(* Logix 5000 project; controller TCP vendor 1 type 14 code 178 rev 35.12; software revision 35.01 *)

TASK MainTask (continuous, watchdog 500 ms) : MainProgram, TCP_Connection
TASK SafetyTask (periodic, rate 20 ms, priority 10, watchdog 20 ms, safety) : SafetyProgram

MODULES
   Local : vendor 1 type 14 code 178 (Compact 0, rev 35.12)
END_MODULES

TYPE MSG_CreateParameters :
STRUCT
   Type : DINT;   // 1 - TCP ; 2 - UPD
   Addr : MSG_SockAddr;   // Address for the Socket
END_STRUCT
END_TYPE

TYPE MSG_OpenConnectionParameters :
STRUCT
   TimeOut : DINT;   // Timeout in milliseconds
   DestAddr : STRING;   // Hostname or IP adress (ex : 10.88.81.10?port=2813 OR name?port=2813)
END_STRUCT
END_TYPE

TYPE MSG_ReadParameters :
STRUCT
   TimeOut : DINT;   // TimeOut in milliseconds
   BufLen : DINT;   // Number of bytes of data to receive
END_STRUCT
END_TYPE

TYPE MSG_ReadResponse :
STRUCT
   FromAddr : MSG_SockAddr;   // A user-defined structure that can contain the address of the device that sends UDP data. This structure is populated from the end device. For TCP or UDP with OpenConnection, this structure is not used and contains all zeros. The TCP connection conveys all remote address information
   BufLen : DINT;   // Contains the number of bytes of data received
   Buf : SINT[484];   // Contains the data. This number must be large enough to contain the maximum amount of data expected. For a standard connection, the maximum is SINT[484]. For a large connection, the maximum is SINT [3984].
END_STRUCT
END_TYPE

TYPE MSG_SockAddr :
STRUCT
   Family : INT;   // Adress Family Must be 2
   Port : INT;   // Port Number - If random needed use 0
   Addr : DINT;   // IP Address - Each Byte are separated for xxx.xxx.xxx.xxx
END_STRUCT
END_TYPE

TYPE MSG_WriteParameters :
STRUCT
   TimeOut : DINT;   // TimeOut in milliseconds
   ToAddr : MSG_SockAddr;   // Structure that contains the address to which to write UDP data. For TCP or UDP with OpenConnection, this structure is not used and contains all zeros. The TCP connection conveys all required remote address information.
   BufLen : DINT;   // Specify the number of bytes of data to write
   Buf : SINT[472];   // Contains the data. This number must be large enough to contain the maximum amount of data expected. For a standard connection, the maximum is SINT[472]. For a large connection, the maximum is SINT [3972].
END_STRUCT
END_TYPE

TYPE UDT_ACTION :   // Action
STRUCT
   Comp : BOOL;   // Action Completed
   OppComp : BOOL;   // Opposite Action Completed
   Clear : BOOL;   // Action is Clear to Go
   Cond_Clear : UDT_ACTION_CLEAR[32];   // Conditions & Texts for Clear (HMI & Supervisor)
   OutPwr : BOOL;   // Output Power For Action
   Cmd : BOOL;   // Action Command
   VirtualOut : BOOL;   // Action Output Request (Virtual )
   Out : BOOL;   // Action Output
   Mem : BOOL;   // Action Memory
   Fault : BOOL;   // Action Faulted
   ActionRequest : BOOL;   // Action Request
END_STRUCT
END_TYPE

TYPE UDT_ACTION_CLEAR :
STRUCT
   Used : BOOL;   // Condition used
   State : BOOL;   // State of the condition
   Text : STRING;   // Text of the condition for HMI & Supervisor
END_STRUCT
END_TYPE

TYPE UDT_BLINK :
STRUCT
   _250ms : BOOL;   // 250ms ON; 250ms OFF
   _500ms : BOOL;   // 500ms ON; 500ms OFF
   _1s : BOOL;   // 1s ON; 1s OFF
   Fast : BOOL;   // Fast Blinking
   Normal : BOOL;   // Normal Blinking
   Edge_1s : BOOL;   // Egde 1s
   Edge_100ms : BOOL;   // Edge 100ms
   Edge_5s : BOOL;   // Edge 5s
END_STRUCT
END_TYPE

TYPE UDT_COOL_DI :
STRUCT
   Load_Presence : BOOL;
   Fan1_CR : BOOL;
   Fan2_CR : BOOL;
END_STRUCT
END_TYPE

TYPE UDT_EDGES :
STRUCT
   Dir_Action : BOOL;   // Direct Action for Raising Edge
   Rev_Action : BOOL;   // Reverse Action for Raising Edge
   Auto_Mode : BOOL;   // Operating Mode Automatic Running for Raising Edge
   Auto_Mode_Switch : BOOL;   // Automatic Mode Switch for Raising Edge
   Manual_Mode_Switch : BOOL;   // Manual Mode Switch for Raising Edge
   Area_Gate_1 : BOOL;   // Area Gate 1 Closed & Locked
   Area_Gate_2 : BOOL;   // Area Gate 2 Closed & Locked
   Area_Gate_3 : BOOL;   // Area Gate 3 Closed & Locked
   Area_Gate_4 : BOOL;   // Area Gate 4 Closed & Locked
   Area_Gate_5 : BOOL;   // Area Gate 5 Closed & Locked
END_STRUCT
END_TYPE

TYPE UDT_FAULT_TREATMENT :
STRUCT
   SAF_DF : INT;   // Faults
   SAF_DF_COPY : INT;   // Fault Copy for Edge Detection
   FAULT_DF : INT[10];   // Faults
   FAULT_COPY : INT[10];   // Fault Copy for Edge Detection
   Level1_Fault_Present : BOOL;   // Level 1 Fault Present
   Level2_Fault_Present : BOOL;   // Level 2 Fault Present
   Level3_Fault_Present : BOOL;   // Level 3 Fault Present
   Level4_Fault_Present : BOOL;   // Level 4 Fault Present
   Fault_Presence : BOOL;   // Fault Presence
   Fault_Appearence : BOOL;   // Fault Appearence
   Treatment_Fault_Copy : BOOL;   // Treatment Fault Copy
   Treatment_Fault_Presence : BOOL;   // Treatment Fault Presence
   Treatment_Fault_Appearence : BOOL;   // Treatment Fault Appearence
END_STRUCT
END_TYPE

TYPE UDT_GEN_ACTION :
STRUCT
   Forcing_Acces_Door : UDT_ACTION;   // Forcing Acces Door for opening
END_STRUCT
END_TYPE

TYPE UDT_GEN_AI :   // Analog Inputs
STRUCT
   Spare : INT;
END_STRUCT
END_TYPE

TYPE UDT_GEN_DELAY :
STRUCT
   Encoding_Req : INT;   // GEN -- Delay Encoding Request
   Encoding_Checksum_Calc_Req : INT;   // GEN -- Delay Encoding Checksum Calculation Request
END_STRUCT
END_TYPE

TYPE UDT_GEN_DELAY_ON :
STRUCT
   Encoding_Req : BOOL;   // GEN -- Delay Encoding Request
   Encoding_Checksum_Calc_Req : BOOL;   // GEN -- Delay Encoding Checksum Calculation Request
END_STRUCT
END_TYPE

TYPE UDT_GEN_DI :   // Digital Inputs
STRUCT
   Reset_EStop : BOOL;   // SBHL19003 : Reset Emergency Stop PB
   Power_ON : BOOL;   // KA8501 : Power ON
   Air_Cond_Temp_OK : BOOL;   // P3601 : Cabinet Air Temperature
   WL_Alarm : BOOL;   // CR241 : Water Loop Alarm Relay
   Auto_Switch : BOOL;   // SB19601 : Selector Auto
   Manual_Switch : BOOL;   // SB19601 : Selector Manu
   Silence_Horn : BOOL;   // SB19602 : Silence Horn
   Reset : BOOL;   // SB19603 : Reset Default
   Reset_Light : BOOL;   // SBHL20702 : Reset Light Curtain
   STORAGE : UDT_STO_DI[64];
   COOL : UDT_COOL_DI[64];
   PC_KTP_Switch : BOOL;   // 0=PC ; 1=KTP
   Direct_Action_Pb : BOOL;   // Direct Action Pushbutton
   Reverse_Action_Pb : BOOL;   // Reverse Action Pushbutton
END_STRUCT
END_TYPE

TYPE UDT_GEN_DO_LIGHT :   // Digital Outputs (Light & Horn)
STRUCT
   Horn : BOOL;   // H24501/H24601 : Horn
   Column_Green : BOOL;   // HL24502/HL24602 : Column Green Light Automatic / Ready
   Column_Red : BOOL;   // HL24503/HL24603 : Column Red Light Critical Event / Fault
   Column_Yellow : BOOL;   // HL24504/HL24604 : Column Yellow Light Manual / Warning
   Column_Blue : BOOL;   // HL24505/HL24605 : Column Blue Light External Help Request
   Column_White : BOOL;   // HL24506/HL24606 : Column White Light Set Up Mode
   Reset_Fault_Light : BOOL;   // PBL19603 : Reset Fault Light
END_STRUCT
END_TYPE

TYPE UDT_GEN_FAULT :
STRUCT
   Gen_Cab_EStop : BOOL;   // Fault : GEN - General Cabinet Estop
   Power_ON : BOOL;   // Fault General Start
   UPS_ON : BOOL;   // Fault UPS ON
   Air_Cond_OK : BOOL;   // Fault Exchanger and Air Temperature Control
   Area_Closed : BOOL;
   PC_EStop : BOOL;   // Fault GEN - Supervisory PC Estop
   UPS_Alarm : BOOL;   // Fault UPS: GEN - UPS Alarm
   UPS_Bat_Disch : BOOL;   // Fault UPS: GEN - Battery is Discharging
   UPS_Batt_Low : BOOL;   // Fault UPS: GEN - Battery Low!!
   UPS_Bypassed : BOOL;   // Fault UPS: GEN - UPS Bypassed
   UPS_Ext_Bypassed : BOOL;   // Fault GEN - External Bypass
   PLC_StopMode : BOOL;   // Fault GEN - PLC in STOP
   Manual_Mode : BOOL;   // Warning: GEN - Periph in Manual Mode
   OPTP_Calculation : BOOL;   // Fault OPTP : Calculation Fault
   OPTP_EL_TR_NRdy : BOOL;   // Fault OPTP EL : Start or Dest Cell not ready for Transfer
   Sfty_Sign_Not_Locked : BOOL;   // Fault GEN - Safety not Locked - Safety Program is not Protected
   Sfty_Sign_Missing : BOOL;   // Fault GEN - Safety Missing Signature - Generate Safety Signature before Locking Task
   Sfty_Sign_Mismatch : BOOL;   // Fault GEN - Safety Signature Mismatch - Safety Program has been Modified
   Com_PC_Loading : BOOL;   // Fault GEN - Communication Fault with PC Supervisory on Loading Side
   Com_PC_Unloading : BOOL;   // Fault GEN - Communication Fault with PC Supervisory on Unloading Side
   Encoding_Error : BOOL;   // Fault GEN - L/U Cell - Encoding Error
   Com_PLC_NANO1 : BOOL;   // Error communication with NANO1
   Com_PLC_NANO2 : BOOL;   // Error communication with NANO2
   Com_PLC_CRYO : BOOL;   // Error communication with CRYO
   Com_PLC_TEMP1 : BOOL;   // Error communication with TEMPER 1
   Com_PLC_TEMP2 : BOOL;   // Error communication with TEMPER 2
   Com_PLC_TEMP3 : BOOL;   // Error communication with TEMPER 3
   Com_PLC_TEMP4 : BOOL;   // Error communication with TEMPER 4
   Com_PLC_TEMP5 : BOOL;   // Error communication with TEMPER 5
   WL_Alarm : BOOL;   // Water Loop : Alarm Relay
   Load_Rejected_Qty_Max : BOOL;   // Load rejected Quantity Max for the Recipe
   Load_Rejected_Qty_Min : BOOL;   // Load rejected Quantity Min for the Recipe
   Load_Rejected_Error_Heat_Recipe : BOOL;   // Load rejected Error in the Step of the Heating Recipe (Temperature must be the same between Ramp and Step after)
   Load_Rejected_Weight_too_heavy : BOOL;   // Load Rejected Error on Total Weight too heavy > 100Kg - 220lbs
   TManager_GetCaution_Error : BOOL;   // T-Manager - GetCaution Request Error
   TManager_GetInstruction_Error : BOOL;   // T-Manager - GetInstruction Request Error
   TManager_TestRunBefore_Error : BOOL;   // T-Manager - Test Run Before Request Error
   TManager_Download_Recipe_Error : BOOL;   // T-Manager - Download Recipe Request Error
   TManager_Insert_Error : BOOL;   // T-Manager - Insert Load Request Error
   TManager_Update_Data_Load_Error : BOOL;   // T-Manager - Update data Load Request Error
   Load_Rejected_Error_Heat_Step_Type : BOOL;   // Load Rejected Error Wrong Type of the Step of the Recipe (Heating cell & Quench )
   Load_Rejected_Miss_Times : BOOL;   // Load Rejected Error Miss times on the Recipe
   Waiting_Transfer_Timeout : BOOL;   // Next order is not in progress - miss conditions
   Miss_Start_Cell_Cond : BOOL;   // Next order is not in progress - Miss Start Cell condition
   Miss_Dest_Cell_Cond : BOOL;   // Next order is not in progress - Miss Dest Cell condition
   Miss_EL_Order_Auth : BOOL;   // Next order is not in progress - Miss Authorization Execution External Loader
END_STRUCT
END_TYPE

TYPE UDT_GEN_FAULT_DELAY :
STRUCT
   Gen_Cab_EStop : INT;   // Fault : GEN - General Cabinet Estop
   Power_ON : INT;   // Fault General Start
   UPS_ON : INT;   // Fault UPS ON
   Air_Cond_OK : INT;   // Fault Exchanger and Air Temperature Control
   Area_Closed : INT;   // Fault GEN - Area Access Door Closed
   PC_EStop : INT;   // Fault GEN - Supervisory PC Estop
   UPS_Alarm : INT;   // Fault UPS: GEN - UPS Alarm
   UPS_Bat_Disch : INT;   // Fault UPS: GEN - Battery is Discharging
   UPS_Batt_Low : INT;   // Fault UPS: GEN - Battery Low!!
   UPS_Bypassed : INT;   // Fault UPS: GEN - UPS Bypassed
   UPS_Ext_Bypassed : INT;   // Fault GEN - External Bypass
   PLC_StopMode : INT;   // Fault GEN - PLC in STOP
   Manual_Mode : INT;   // Warning: GEN - Nano in Manual Mode
   OPTP_Calculation : INT;   // Fault OPTP : Calculation Fault
   OPTP_EL_TR_NRdy : INT;   // Fault OPTP EL : Start or Dest Cell not ready for Transfer
   Sfty_Sign_Not_Locked : INT;   // Fault GEN - Safety not Locked - Safety Program is not Protected
   Sfty_Sign_Missing : INT;   // Fault GEN - Safety Missing Signature - Generate Safety Signature before Locking Task
   Sfty_Sign_Mismatch : INT;   // Fault GEN - Safety Signature Mismatch - Safety Program has been Modified
   Com_PC_Loading : INT;   // Fault GEN - Communication Fault with PC Supervisory on Loading Side
   Com_PC_Unloading : INT;   // Fault GEN - Communication Fault with PC Supervisory on Unloading Side
   Encoding_Error : INT;   // Fault GEN - L/U Cell - Encoding Error
   Com_Error_Send_Load_PLC_NANO1 : INT;   // Fault GEN - Error on the Send data for Load to the NANO1
   Timeout_Recv_Cyclic_PLC_NANO1 : INT;   // Fault GEN - Time out receiving data from PLC NANO1
   Com_Error_Send_Load_PLC_NANO2 : INT;   // Fault GEN - Error on the Send data for Load to the NANO2
   Timeout_Recv_Cyclic_PLC_NANO2 : INT;   // Fault GEN - Time out receiving data from PLC NANO2
   WL_Alarm : INT;
END_STRUCT
END_TYPE

TYPE UDT_GEN_FAULT_ETHIP :
STRUCT
   RemIO : BOOL;   // Ethernet IP : Rem IO
   x1 : BOOL;
   x2 : BOOL;
   x3 : BOOL;
   x4 : BOOL;
   E12401_MAIN : BOOL;
   E12501_MAIN : BOOL;
   X26001_MAIN : BOOL;   // Ethernet IP : X26001-Armblock
   X26002_MAIN : BOOL;   // Ethernet IP : X26001-Armblock
   X26101_MAIN : BOOL;   // Ethernet IP : X26101-Armblock
   X26201_MAIN : BOOL;   // Ethernet IP : X26201-Armblock
   X26301_MAIN : BOOL;   // Ethernet IP : X26301-Armblock
   X26401_MAIN : BOOL;   // Ethernet IP : X26401-Armblock (Water Loop)
   A6001_MAIN : BOOL;   // Ethernet IP : VFD A6001 - External Loader - Translation
   A6101_MAIN : BOOL;   // Ethernet IP : VFD A6001 - External Loader - Forks
   A6201_MAIN : BOOL;   // Ethernet IP : VFD A6001 - External Loader - Lifting
   A11201_FORTRESS : BOOL;   // Ethernet IP : FORTRESS A11201
   A11301_FORTRESS : BOOL;   // Ethernet IP : FORTRESS A11301
   E14201_STRATIX : BOOL;
   X26301_WL : BOOL;   // Ethernet IP : X26001-Armblock (Water Loop)
   Nano1 : BOOL;   // Ethernet IP : PLC Nano1
   Nano2 : BOOL;   // Ethernet IP : PLC Nano 2
   Cryo : BOOL;   // Ethernet IP : PLC Cryo
   Temper1 : BOOL;   // Ethernet IP : PLC Temper 1
   Temper2 : BOOL;   // Ethernet IP : PLC Temper 2
   Temper3 : BOOL;   // Ethernet IP : PLC Temper 3
   Temper4 : BOOL;   // Ethernet IP : PLC Temper 4
END_STRUCT
END_TYPE

TYPE UDT_GEN_FAULT_SAFETY :
STRUCT
   Estop : BOOL;   // GEN -EStop OK
   MCRA_ON : BOOL;   // GEN - MCR 1A/2A (Emergency Stop)
   SCRA_ON : BOOL;   // GEN - SCR 1A/2A
   SCRB_ON : BOOL;   // GEN - SCR 1B/2B
   SCRC_ON : BOOL;   // GEN - SCR 1C/2C
   Sfty_Ack_Req : BOOL;   // GEN Fault -- Safety Acknowledge Requested
END_STRUCT
END_TYPE

TYPE UDT_GEN_INFO :
STRUCT
   Normal_Supply : BOOL;   // GEN -- Normal Supply
   UPS_Supply : BOOL;   // GEN -- Saved Supply
   Normal_Volt_Flt_Mem : BOOL;   // GEN -- Normal Voltage presence Fault Memory
   KTP_Manual_Cmd_Auth : BOOL;   // GEN -- KTP Manual Command Authorization
   Init_Cond : BOOL;   // GEN -- Initial Conditions for Auto Mode
   Out_Oper_Mode : BOOL;   // GEN -- Conditions for Switching to Out of Operation Mode
   Stop_Oper_Mode : BOOL;   // GEN -- Stop Operation Mode
   No_Motion_for_Door_Access : BOOL;   // GEN - No Motion for Door Access
   No_Motion_EL : BOOL;   // External Loader : No motion
   No_Motion_LD : BOOL;   // Loading : No Motion
   No_Motion_UL : BOOL;   // Unloading : No Motion
   No_Motion_Cool : BOOL;   // Cooling : No Motion
   No_Motion_NANO : BOOL;   // NANO : No Motion (By dialogue)
   No_Motion_TEMP : BOOL;   // TEMPER : No Motion (By dialogue)
   No_Motion_CRYO : BOOL;   // CRYO : No Motion (By dialogue)
   Access_Request : BOOL;   // Request for access to the outer peripheral zone
   Access_Authorized : BOOL;   // Acces Authorized
   Access_OK : BOOL;   // Acces OK : Solenoid Active
   Cond_Auto_Mode : UDT_ACTION;   // Init Conditions for Auto Mode
   Cond_Auto_Mode_State : DINT;   // state for supervisory
   Cond_Auto_Mode_Used : DINT;   // Used for Supervisory
END_STRUCT
END_TYPE

TYPE UDT_GEN_MEAS :
STRUCT
   Spare : REAL;
END_STRUCT
END_TYPE

TYPE UDT_GEN_RUNNING_TIME :
STRUCT
   Spare : DINT;
END_STRUCT
END_TYPE

TYPE UDT_ID_READER :
STRUCT
   INPUT : UDT_ID_READER_IN;
   OUTPUT : UDT_ID_READER_OUT;
END_STRUCT
END_TYPE

TYPE UDT_ID_READER_IN :
STRUCT
   Sequence_Low : SINT;
   Sequence_High : SINT;
   LUID_Low : SINT;
   LUID_High : SINT;
   Bit_Counf_of_ID : SINT;
   Zero_Padding : SINT;
   ID_Data_bytes : SINT[32];
END_STRUCT
END_TYPE

TYPE UDT_ID_READER_OUT :
STRUCT
   Led_Control : BOOL;
   Beep : BOOL;
END_STRUCT
END_TYPE

TYPE UDT_OPERATING_MODE :
STRUCT
   Out_of_Operation : BOOL;   // Out of Operation Mode
   Init_Missing_Cond : BOOL;   // Operating Mode Initiales Conditions Missing
   Origin : BOOL;   // Operating Mode Origine
   Waiting_Cycle_Start : BOOL;   // Operating Mode Waiting for Cycle Start
   Manual : BOOL;   // Operating Mode Manual
   Auto : BOOL;   // Operating Mode Automatic Running
END_STRUCT
END_TYPE

TYPE UDT_OPTP_BUFFER :
STRUCT
   Buffer : SINT[5000];
   Lenght : DINT;
   New_Data : BOOL;
END_STRUCT
END_TYPE

TYPE UDT_OPTP_RECV_CONTROL :
STRUCT
   New_TCP_Data : BOOL;
   New_Frame_Complete : BOOL;
END_STRUCT
END_TYPE

TYPE UDT_STO_DI :
STRUCT
   Load_Presence_Physical : BOOL;   // Physical Presence on Storage
END_STRUCT
END_TYPE

VAR_GLOBAL   (* controller tags *)
   Destination_Element_Read_Request : MSG_ReadResponse := (FromAddr.Family := 2, Buf[0] := 107, Buf[1] := 99, Buf[2] := 111, Buf[9] := 1, Buf[12] := 107, Buf[13] := 99, Buf[14] := 111, Buf[21] := 3, Buf[25] := 1, Buf[29] := 1, Buf[34] := 15, Buf[35] := -125, Buf[36] := -20, Buf[37] := -78, Buf[38] := 50, Buf[39] := 54, Buf[40] := 48, Buf[41] := 51, Buf[42] := 48, Buf[43] := 52, Buf[44] := 48, Buf[45] := 53, Buf[46] := 48, Buf[61] := 3, Buf[63] := -115, Buf[64] := 23, Buf[65] := 112, Buf[66] := 19, Buf[67] := -119, Buf[75] := 48, Buf[76] := 7, Buf[77] := -47, Buf[79] := 60, Buf[80] := 107, Buf[81] := 99, Buf[82] := 111, Buf[89] := 3, Buf[91] := 1, Buf[92] := -20, Buf[93] := -95, Buf[94] := 50, Buf[95] := 54, Buf[96] := 48, Buf[97] := 51, Buf[98] := 48, Buf[99] := 52, Buf[100] := 48, Buf[101] := 51, Buf[102] := 51, Buf[117] := 93, Buf[119] := -115, Buf[120] := 2, Buf[121] := 89, Buf[122] := 19, Buf[123] := -119, Buf[126] := 4, Buf[127] := -52, Buf[130] := 5, Buf[131] := 8,
        Buf[132] := 7, Buf[133] := -41, Buf[135] := 60, Buf[136] := 107, Buf[137] := 99, Buf[138] := 111, Buf[145] := 3, Buf[147] := 2, Buf[148] := 107, Buf[149] := 99, Buf[150] := 111, Buf[157] := 3, Buf[159] := 2, Buf[160] := -20, Buf[161] := -95, Buf[162] := 50, Buf[163] := 54, Buf[164] := 48, Buf[165] := 51, Buf[166] := 48, Buf[167] := 52, Buf[168] := 48, Buf[169] := 51, Buf[170] := 51, Buf[185] := 93, Buf[187] := -115, Buf[188] := 2, Buf[189] := 89, Buf[190] := 19, Buf[191] := -119, Buf[194] := 5, Buf[195] := 59, Buf[198] := 5, Buf[199] := 119, Buf[200] := 7, Buf[201] := -41, Buf[203] := 60, Buf[204] := 107, Buf[205] := 99, Buf[206] := 111, Buf[213] := 3, Buf[215] := 3, Buf[216] := 107, Buf[217] := 99, Buf[218] := 111, Buf[225] := 3, Buf[227] := 3, Buf[229] := 4, Buf[233] := 4, Buf[238] := 15, Buf[239] := -125, Buf[240] := -20, Buf[241] := -95, Buf[242] := 50, Buf[243] := 54, Buf[244] := 48, Buf[245] := 51, Buf[246] := 48, Buf[247] := 52, Buf[248] := 48,
        Buf[249] := 51, Buf[250] := 51, Buf[265] := 93, Buf[267] := -115, Buf[268] := 2, Buf[269] := 89, Buf[270] := 19, Buf[271] := -119, Buf[274] := 9, Buf[275] := -13, Buf[278] := 10, Buf[279] := 47, Buf[280] := 7, Buf[281] := -41, Buf[283] := 60, Buf[284] := 107, Buf[285] := 99, Buf[286] := 111, Buf[293] := 3, Buf[295] := 4, Buf[297] := 5, Buf[301] := 5, Buf[306] := 15, Buf[307] := -125, Buf[308] := -20, Buf[309] := -95, Buf[310] := 50, Buf[311] := 54, Buf[312] := 48, Buf[313] := 51, Buf[314] := 48, Buf[315] := 52, Buf[316] := 48, Buf[317] := 51, Buf[318] := 51, Buf[333] := 93, Buf[335] := -115, Buf[336] := 2, Buf[337] := 89, Buf[338] := 19, Buf[339] := -119, Buf[342] := 13, Buf[343] := -50, Buf[346] := 14, Buf[347] := 10, Buf[348] := 7, Buf[349] := -41, Buf[351] := 60, Buf[352] := 107, Buf[353] := 99, Buf[354] := 111, Buf[361] := 3, Buf[363] := 5, Buf[365] := 6, Buf[369] := 6, Buf[374] := 15, Buf[375] := -125, Buf[376] := -20, Buf[377] := -95, Buf[378] := 50,
        Buf[379] := 54, Buf[380] := 48, Buf[381] := 51, Buf[382] := 48, Buf[383] := 52, Buf[384] := 48, Buf[385] := 51, Buf[386] := 51, Buf[401] := 93, Buf[403] := -115, Buf[404] := 2, Buf[405] := 89, Buf[406] := 19, Buf[407] := -119, Buf[410] := 14, Buf[411] := 25, Buf[414] := 14, Buf[415] := 85, Buf[416] := 7, Buf[417] := -41, Buf[419] := 60, Buf[420] := 107, Buf[421] := 99, Buf[422] := 111, Buf[429] := 3, Buf[431] := 6, Buf[433] := 7, Buf[437] := 7, Buf[442] := 15, Buf[443] := -125, Buf[444] := -20, Buf[445] := -95, Buf[446] := 50, Buf[447] := 54, Buf[448] := 48, Buf[449] := 51, Buf[450] := 48, Buf[451] := 52, Buf[452] := 48, Buf[453] := 51, Buf[454] := 51, Buf[469] := 93, Buf[471] := -115, Buf[472] := 2, Buf[473] := 89, Buf[474] := 19, Buf[475] := -119, Buf[478] := 15, Buf[479] := -31, Buf[482] := 16, Buf[483] := 29);
   Destination_Element_Write_Request : DINT := 48;   // Lenght of the Data written
   Instance_OPTP : DINT := 21276;
   MSG_Create_Socket : MESSAGE;
        MessageParameters(ServiceCode := 16#004b, LocalElement := Source_Element_Create_Socket, DestinationTag := Instance_OPTP, ...)
   MSG_Delete_All_Socket : MESSAGE;
        MessageParameters(ServiceCode := 16#0051, ...)
   MSG_Open_Connection : MESSAGE;
        MessageParameters(ServiceCode := 16#004c, LocalElement := Source_Element_Open_Connection, ...)
   MSG_Read_Request : MESSAGE;
        MessageParameters(ServiceCode := 16#004d, LocalElement := Source_Element_Read_Request, DestinationTag := Destination_Element_Read_Request, ...)
   MSG_Write_Request : MESSAGE;
        MessageParameters(ServiceCode := 16#004e, LocalElement := Source_Element_Write_Request, DestinationTag := Destination_Element_Write_Request, ...)
   Source_Element_Create_Socket : MSG_CreateParameters := (Type := 1, Addr.Family := 2, Addr.Port := 10002);   // Source parameters for MSG Create Socket
   Source_Element_Open_Connection : MSG_OpenConnectionParameters := (TimeOut := 5000, DestAddr := '192.120.0.203?port=5010$00');
   Source_Element_Read_Request : MSG_ReadParameters := (TimeOut := 3000, BufLen := 484);
   Source_Element_Write_Request : MSG_WriteParameters := (TimeOut := 5000, BufLen := 1, Buf[0] := 104, Buf[1] := 101, Buf[2] := 108, Buf[3] := 108, Buf[4] := 111);
END_VAR

PROGRAM MainProgram   (* main routine MainRoutine *)

ROUTINE MainRoutine   (* ladder *)
END_ROUTINE
END_PROGRAM

PROGRAM SafetyProgram   (* main routine MainRoutine, safety *)

ROUTINE MainRoutine   (* ladder *)
END_ROUTINE
END_PROGRAM

PROGRAM TCP_Connection   (* main routine Main *)
VAR
   buff_ind : DINT;
   Buff_ok : BOOL;
   Check_Buflenght : BOOL;
   Connection_Ok : BOOL := 1;
   Element_Read_buffer : SINT[5000];
   ind : DINT := 1;
   ONS : BOOL[32];
   Open_started : BOOL;
   OPTP_Data_RCV : UDT_OPTP_BUFFER := (Buffer[0] := 107, Buffer[1] := 99, Buffer[2] := 111, Buffer[9] := 3, Buffer[12] := 107, Buffer[13] := 99, Buffer[14] := 111, Buffer[21] := 3, Buffer[24] := -20, Buffer[25] := -78, Buffer[26] := 50, Buffer[27] := 54, Buffer[28] := 48, Buffer[29] := 51, Buffer[30] := 48, Buffer[31] := 52, Buffer[32] := 48, Buffer[33] := 53, Buffer[34] := 48, Buffer[49] := 3, Buffer[51] := -115, Buffer[52] := 23, Buffer[53] := 112, Buffer[54] := 19, Buffer[55] := -119, Buffer[63] := 48, Buffer[64] := 7, Buffer[65] := -47, Buffer[67] := 60, Buffer[68] := 107, Buffer[69] := 99, Buffer[70] := 111, Buffer[77] := 3, Buffer[79] := 1, Buffer[80] := 107, Buffer[81] := 99, Buffer[82] := 111, Buffer[89] := 3, Buffer[91] := 1, Buffer[92] := -20, Buffer[93] := -95, Buffer[94] := 50, Buffer[95] := 54, Buffer[96] := 48, Buffer[97] := 51, Buffer[98] := 48, Buffer[99] := 52, Buffer[100] := 48, Buffer[101] := 51, Buffer[102] := 51, Buffer[117] := 93, Buffer[119] := -115, Buffer[120] := 2, Buffer[121] := 89, Buffer[122] := 19, Buffer[123] := -119, Buffer[126] := 4, Buffer[127] := -52, Buffer[130] := 5, Buffer[131] := 8,
        Buffer[132] := 7, Buffer[133] := -41, Buffer[135] := 60, Buffer[136] := 107, Buffer[137] := 99, Buffer[138] := 111, Buffer[145] := 3, Buffer[147] := 2, Buffer[148] := 107, Buffer[149] := 99, Buffer[150] := 111, Buffer[157] := 3, Buffer[159] := 2, Buffer[160] := -20, Buffer[161] := -95, Buffer[162] := 50, Buffer[163] := 54, Buffer[164] := 48, Buffer[165] := 51, Buffer[166] := 48, Buffer[167] := 52, Buffer[168] := 48, Buffer[169] := 51, Buffer[170] := 51, Buffer[185] := 93, Buffer[187] := -115, Buffer[188] := 2, Buffer[189] := 89, Buffer[190] := 19, Buffer[191] := -119, Buffer[194] := 5, Buffer[195] := 59, Buffer[198] := 5, Buffer[199] := 119, Buffer[200] := 7, Buffer[201] := -41, Buffer[203] := 60, Buffer[204] := 107, Buffer[205] := 99, Buffer[206] := 111, Buffer[213] := 3, Buffer[215] := 3, Buffer[216] := 107, Buffer[217] := 99, Buffer[218] := 111, Buffer[225] := 3, Buffer[227] := 3, Buffer[228] := -20, Buffer[229] := -95, Buffer[230] := 50, Buffer[231] := 54, Buffer[232] := 48, Buffer[233] := 51, Buffer[234] := 48, Buffer[235] := 52, Buffer[236] := 48, Buffer[237] := 51, Buffer[238] := 51, Buffer[253] := 93, Buffer[255] := -115,
        Buffer[256] := 2, Buffer[257] := 89, Buffer[258] := 19, Buffer[259] := -119, Buffer[262] := 9, Buffer[263] := -13, Buffer[266] := 10, Buffer[267] := 47, Buffer[268] := 7, Buffer[269] := -41, Buffer[271] := 60, Buffer[272] := 107, Buffer[273] := 99, Buffer[274] := 111, Buffer[281] := 3, Buffer[283] := 4, Buffer[284] := 107, Buffer[285] := 99, Buffer[286] := 111, Buffer[293] := 3, Buffer[295] := 4, Buffer[296] := -20, Buffer[297] := -95, Buffer[298] := 50, Buffer[299] := 54, Buffer[300] := 48, Buffer[301] := 51, Buffer[302] := 48, Buffer[303] := 52, Buffer[304] := 48, Buffer[305] := 51, Buffer[306] := 51, Buffer[321] := 93, Buffer[323] := -115, Buffer[324] := 2, Buffer[325] := 89, Buffer[326] := 19, Buffer[327] := -119, Buffer[330] := 13, Buffer[331] := -50, Buffer[334] := 14, Buffer[335] := 10, Buffer[336] := 7, Buffer[337] := -41, Buffer[339] := 60, Buffer[340] := 107, Buffer[341] := 99, Buffer[342] := 111, Buffer[349] := 3, Buffer[351] := 5, Buffer[352] := 107, Buffer[353] := 99, Buffer[354] := 111, Buffer[361] := 3, Buffer[363] := 5, Buffer[364] := -20, Buffer[365] := -95, Buffer[366] := 50, Buffer[367] := 54, Buffer[368] := 48,
        Buffer[369] := 51, Buffer[370] := 48, Buffer[371] := 52, Buffer[372] := 48, Buffer[373] := 51, Buffer[374] := 51, Buffer[389] := 93, Buffer[391] := -115, Buffer[392] := 2, Buffer[393] := 89, Buffer[394] := 19, Buffer[395] := -119, Buffer[398] := 14, Buffer[399] := 25, Buffer[402] := 14, Buffer[403] := 85, Buffer[404] := 7, Buffer[405] := -41, Buffer[407] := 60, Buffer[410] := 14, Buffer[411] := 25, Buffer[414] := 14, Buffer[415] := 85, Buffer[416] := 7, Buffer[417] := -41, Buffer[419] := 60, Buffer[420] := 107, Buffer[421] := 99, Buffer[422] := 111, Buffer[429] := 3, Buffer[431] := 6, Buffer[432] := -20, Buffer[433] := -95, Buffer[434] := 50, Buffer[435] := 54, Buffer[436] := 48, Buffer[437] := 51, Buffer[438] := 48, Buffer[439] := 52, Buffer[440] := 48, Buffer[441] := 51, Buffer[442] := 51, Buffer[457] := 93, Buffer[459] := -115, Buffer[460] := 2, Buffer[461] := 89, Buffer[462] := 19, Buffer[463] := -119, Buffer[466] := 15, Buffer[467] := -31, Buffer[470] := 16, Buffer[471] := 29, Buffer[472] := 7, Buffer[473] := -41, Buffer[475] := 60, Buffer[478] := 15, Buffer[479] := -31, Buffer[482] := 16, Buffer[483] := 29, Buffer[484] := 7,
        Buffer[485] := -41, Buffer[487] := 60, Buffer[489] := 8, Buffer[493] := 8, Buffer[498] := 15, Buffer[499] := -125, Buffer[500] := -20, Buffer[501] := -95, Buffer[502] := 50, Buffer[503] := 54, Buffer[504] := 48, Buffer[505] := 51, Buffer[506] := 48, Buffer[507] := 52, Buffer[508] := 48, Buffer[509] := 51, Buffer[510] := 51, Buffer[525] := 93, Buffer[527] := -115, Buffer[528] := 2, Buffer[529] := 89, Buffer[530] := 19, Buffer[531] := -119, Buffer[534] := 16, Buffer[535] := 65, Buffer[538] := 16, Buffer[539] := 125, Buffer[540] := 7, Buffer[541] := -41, Buffer[543] := 60, Buffer[544] := 107, Buffer[545] := 99, Buffer[546] := 111, Buffer[553] := 3, Buffer[555] := 8, Buffer[557] := 9, Buffer[561] := 9, Buffer[566] := 15, Buffer[567] := -125, Buffer[568] := -20, Buffer[569] := -95, Buffer[570] := 50, Buffer[571] := 54, Buffer[572] := 48, Buffer[573] := 51, Buffer[574] := 48, Buffer[575] := 52, Buffer[576] := 48, Buffer[577] := 51, Buffer[578] := 51, Buffer[593] := 93, Buffer[595] := -115, Buffer[596] := 2, Buffer[597] := 89, Buffer[598] := 19, Buffer[599] := -119, Buffer[602] := 16, Buffer[603] := -116, Buffer[606] := 16, Buffer[607] := -56,
        Buffer[608] := 7, Buffer[609] := -41, Buffer[611] := 60, Buffer[612] := 107, Buffer[613] := 99, Buffer[614] := 111, Buffer[621] := 3, Buffer[623] := 9, Buffer[624] := 107, Buffer[625] := 99, Buffer[626] := 111, Buffer[633] := 3, Buffer[635] := 9, Buffer[636] := -20, Buffer[637] := -95, Buffer[638] := 50, Buffer[639] := 54, Buffer[640] := 48, Buffer[641] := 51, Buffer[642] := 48, Buffer[643] := 52, Buffer[644] := 48, Buffer[645] := 51, Buffer[646] := 51, Buffer[661] := 93, Buffer[663] := -115, Buffer[664] := 2, Buffer[665] := 89, Buffer[666] := 19, Buffer[667] := -119, Buffer[670] := 18, Buffer[671] := -58, Buffer[674] := 19, Buffer[675] := 2, Buffer[676] := 7, Buffer[677] := -41, Buffer[679] := 60, Buffer[680] := 107, Buffer[681] := 99, Buffer[682] := 111, Buffer[689] := 3, Buffer[691] := 12, Buffer[693] := 12, Buffer[697] := 12, Buffer[702] := 15, Buffer[703] := -125, Buffer[704] := -20, Buffer[705] := -95, Buffer[706] := 50, Buffer[707] := 54, Buffer[708] := 48, Buffer[709] := 51, Buffer[710] := 48, Buffer[711] := 52, Buffer[712] := 48, Buffer[713] := 51, Buffer[714] := 51, Buffer[729] := 93, Buffer[731] := -115, Buffer[732] := 2,
        Buffer[733] := 89, Buffer[734] := 19, Buffer[735] := -119, Buffer[738] := 18, Buffer[739] := -58, Buffer[742] := 19, Buffer[743] := 2, Buffer[744] := 7, Buffer[745] := -41, Buffer[747] := 60, Buffer[748] := 107, Buffer[749] := 99, Buffer[750] := 111, Buffer[757] := 3, Buffer[759] := 12, Buffer[761] := 12, Buffer[765] := 12, Buffer[770] := 15, Buffer[771] := -125, Buffer[772] := -20, Buffer[773] := -95, Buffer[774] := 50, Buffer[775] := 54, Buffer[776] := 48, Buffer[777] := 51, Buffer[778] := 48, Buffer[779] := 52, Buffer[780] := 48, Buffer[781] := 51, Buffer[782] := 51, Buffer[797] := 93, Buffer[799] := -115, Buffer[800] := 2, Buffer[801] := 89, Buffer[802] := 19, Buffer[803] := -119, Buffer[806] := 18, Buffer[807] := -58, Buffer[810] := 19, Buffer[811] := 2, Buffer[812] := 7, Buffer[813] := -41, Buffer[815] := 60, Buffer[816] := 107, Buffer[817] := 99, Buffer[818] := 111, Buffer[825] := 3, Buffer[827] := 12, Buffer[829] := 13, Buffer[833] := 13, Buffer[838] := 15, Buffer[839] := -125, Buffer[840] := -20, Buffer[841] := -95, Buffer[842] := 50, Buffer[843] := 54, Buffer[844] := 48, Buffer[845] := 51, Buffer[846] := 48, Buffer[847] := 52,
        Buffer[848] := 48, Buffer[849] := 51, Buffer[850] := 51, Buffer[865] := 93, Buffer[867] := -115, Buffer[868] := 2, Buffer[869] := 89, Buffer[870] := 19, Buffer[871] := -119, Buffer[874] := 19, Buffer[875] := 57, Buffer[878] := 19, Buffer[879] := 117, Buffer[880] := 7, Buffer[881] := -41, Buffer[883] := 60, Buffer[884] := 107, Buffer[885] := 99, Buffer[886] := 111, Buffer[893] := 3, Buffer[895] := 13, Buffer[897] := 14, Buffer[901] := 14, Buffer[906] := 15, Buffer[907] := -125, Buffer[908] := -20, Buffer[909] := -95, Buffer[910] := 50, Buffer[911] := 54, Buffer[912] := 48, Buffer[913] := 51, Buffer[914] := 48, Buffer[915] := 52, Buffer[916] := 48, Buffer[917] := 51, Buffer[918] := 51, Buffer[933] := 64, Buffer[935] := 93, Buffer[936] := 1, Buffer[937] := -12, Buffer[938] := 2, Buffer[939] := 89, Buffer[942] := 15, Buffer[943] := 17, Buffer[946] := 15, Buffer[947] := 77, Buffer[948] := 7, Buffer[949] := -42, Buffer[951] := 60, Buffer[954] := 15, Buffer[955] := 12, Buffer[958] := 15, Buffer[959] := 72, Buffer[960] := 7, Buffer[961] := -43, Buffer[963] := 60, Buffer[965] := 18, Buffer[969] := 18, Buffer[974] := 15, Buffer[975] := -125,
        Buffer[976] := -20, Buffer[977] := -95, Buffer[978] := 50, Buffer[979] := 54, Buffer[980] := 48, Buffer[981] := 51, Buffer[982] := 48, Buffer[983] := 52, Buffer[984] := 48, Buffer[985] := 51, Buffer[986] := 51, Buffer[1001] := 93, Buffer[1003] := -115, Buffer[1004] := 2, Buffer[1005] := 89, Buffer[1006] := 19, Buffer[1007] := -119, Buffer[1010] := 22, Buffer[1011] := -28, Buffer[1014] := 23, Buffer[1015] := 32, Buffer[1016] := 7, Buffer[1017] := -41, Buffer[1019] := 60, Buffer[1020] := 107, Buffer[1021] := 99, Buffer[1022] := 111, Buffer[1029] := 3, Buffer[1031] := 18, Buffer[1033] := 18, Buffer[1037] := 18, Buffer[1042] := 15, Buffer[1043] := -125, Buffer[1044] := -20, Buffer[1045] := -95, Buffer[1046] := 50, Buffer[1047] := 54, Buffer[1048] := 48, Buffer[1049] := 51, Buffer[1050] := 48, Buffer[1051] := 52, Buffer[1052] := 48, Buffer[1053] := 51, Buffer[1054] := 51, Buffer[1069] := 93, Buffer[1071] := -115, Buffer[1072] := 2, Buffer[1073] := 89, Buffer[1074] := 19, Buffer[1075] := -119, Buffer[1078] := 22, Buffer[1079] := -28, Buffer[1082] := 23, Buffer[1083] := 32, Buffer[1084] := 7, Buffer[1085] := -41, Buffer[1087] := 60, Buffer[1088] := 107, Buffer[1089] := 99, Buffer[1090] := 111,
        Buffer[1097] := 3, Buffer[1099] := 18, Buffer[1101] := 18, Buffer[1105] := 18, Buffer[1110] := 15, Buffer[1111] := -125, Buffer[1112] := -20, Buffer[1113] := -95, Buffer[1114] := 50, Buffer[1115] := 54, Buffer[1116] := 48, Buffer[1117] := 51, Buffer[1118] := 48, Buffer[1119] := 52, Buffer[1120] := 48, Buffer[1121] := 51, Buffer[1122] := 51, Buffer[1137] := 93, Buffer[1139] := -115, Buffer[1140] := 2, Buffer[1141] := 89, Buffer[1142] := 19, Buffer[1143] := -119, Buffer[1146] := 22, Buffer[1147] := -28, Buffer[1150] := 23, Buffer[1151] := 32, Buffer[1152] := 7, Buffer[1153] := -41, Buffer[1155] := 60, Buffer[1156] := 107, Buffer[1157] := 99, Buffer[1158] := 111, Buffer[1165] := 3, Buffer[1167] := 18, Buffer[1169] := 18, Buffer[1173] := 18, Buffer[1178] := 15, Buffer[1179] := -125, Buffer[1180] := -20, Buffer[1181] := -95, Buffer[1182] := 50, Buffer[1183] := 54, Buffer[1184] := 48, Buffer[1185] := 51, Buffer[1186] := 48, Buffer[1187] := 52, Buffer[1188] := 48, Buffer[1189] := 51, Buffer[1190] := 51, Buffer[1205] := 93, Buffer[1207] := -115, Buffer[1208] := 2, Buffer[1209] := 89, Buffer[1210] := 19, Buffer[1211] := -119, Buffer[1214] := 22, Buffer[1215] := -28, Buffer[1218] := 23, Buffer[1219] := 32,
        Buffer[1220] := 7, Buffer[1221] := -41, Buffer[1223] := 60, Buffer[1224] := 107, Buffer[1225] := 99, Buffer[1226] := 111, Buffer[1233] := 3, Buffer[1235] := 18, Buffer[1237] := 24, Buffer[1241] := 24, Buffer[1246] := 15, Buffer[1247] := -125, Buffer[1248] := -20, Buffer[1249] := -95, Buffer[1250] := 50, Buffer[1251] := 54, Buffer[1252] := 48, Buffer[1253] := 51, Buffer[1254] := 48, Buffer[1255] := 52, Buffer[1256] := 48, Buffer[1257] := 51, Buffer[1258] := 51, Buffer[1273] := 93, Buffer[1275] := -115, Buffer[1276] := 2, Buffer[1277] := 89, Buffer[1278] := 19, Buffer[1279] := -119, Buffer[1282] := 27, Buffer[1283] := 87, Buffer[1286] := 27, Buffer[1287] := -109, Buffer[1288] := 7, Buffer[1289] := -41, Buffer[1291] := 60, Buffer[1292] := 107, Buffer[1293] := 99, Buffer[1294] := 111, Buffer[1301] := 3, Buffer[1303] := 24, Buffer[1305] := 20, Buffer[1309] := 20, Buffer[1314] := 15, Buffer[1315] := -125, Buffer[1316] := -20, Buffer[1317] := -97, Buffer[1318] := 50, Buffer[1319] := 54, Buffer[1320] := 48, Buffer[1321] := 51, Buffer[1322] := 48, Buffer[1323] := 52, Buffer[1324] := 48, Buffer[1325] := 51, Buffer[1326] := 49, Buffer[1341] := 63, Buffer[1343] := 95, Buffer[1344] := 1, Buffer[1345] := -12,
        Buffer[1346] := 2, Buffer[1347] := 88, Buffer[1350] := 14, Buffer[1351] := 87, Buffer[1354] := 14, Buffer[1355] := -109, Buffer[1356] := 7, Buffer[1357] := -44, Buffer[1359] := 60, Buffer[1360] := 107, Buffer[1361] := 99, Buffer[1362] := 111, Buffer[1369] := 3, Buffer[1371] := 24, Buffer[1373] := 25, Buffer[1377] := 25, Buffer[1382] := 15, Buffer[1383] := -125, Buffer[1384] := -20, Buffer[1385] := -95, Buffer[1386] := 50, Buffer[1387] := 54, Buffer[1388] := 48, Buffer[1389] := 51, Buffer[1390] := 48, Buffer[1391] := 52, Buffer[1392] := 48, Buffer[1393] := 51, Buffer[1394] := 51, Buffer[1409] := 93, Buffer[1411] := -115, Buffer[1412] := 2, Buffer[1413] := 89, Buffer[1414] := 19, Buffer[1415] := -119, Buffer[1418] := 29, Buffer[1419] := -75, Buffer[1422] := 29, Buffer[1423] := -15, Buffer[1424] := 7, Buffer[1425] := -41, Buffer[1427] := 60, Buffer[1428] := 107, Buffer[1429] := 99, Buffer[1430] := 111, Buffer[1437] := 3, Buffer[1439] := 25, Buffer[1441] := 25, Buffer[1445] := 25, Buffer[1450] := 15, Buffer[1451] := -125, Buffer[1452] := -20, Buffer[1453] := -95, Buffer[1454] := 50, Buffer[1455] := 54, Buffer[1456] := 48, Buffer[1457] := 51, Buffer[1458] := 48, Buffer[1459] := 52, Buffer[1460] := 48,
        Buffer[1461] := 51, Buffer[1462] := 51, Buffer[1477] := 93, Buffer[1479] := -115, Buffer[1480] := 2, Buffer[1481] := 89, Buffer[1482] := 19, Buffer[1483] := -119, Buffer[1486] := 29, Buffer[1487] := -75, Buffer[1490] := 29, Buffer[1491] := -15, Buffer[1492] := 7, Buffer[1493] := -41, Buffer[1495] := 60, Buffer[1496] := 107, Buffer[1497] := 99, Buffer[1498] := 111, Buffer[1505] := 3, Buffer[1507] := 25, Buffer[1509] := 25, Buffer[1513] := 25, Buffer[1518] := 15, Buffer[1519] := -125, Buffer[1520] := -20, Buffer[1521] := -95, Buffer[1522] := 50, Buffer[1523] := 54, Buffer[1524] := 48, Buffer[1525] := 51, Buffer[1526] := 48, Buffer[1527] := 52, Buffer[1528] := 48, Buffer[1529] := 51, Buffer[1530] := 51, Buffer[1545] := 93, Buffer[1547] := -115, Buffer[1548] := 2, Buffer[1549] := 89, Buffer[1550] := 19, Buffer[1551] := -119, Buffer[1554] := 29, Buffer[1555] := -75, Buffer[1558] := 29, Buffer[1559] := -15, Buffer[1560] := 7, Buffer[1561] := -41, Buffer[1563] := 60, Buffer[1564] := 107, Buffer[1565] := 99, Buffer[1566] := 111, Buffer[1573] := 3, Buffer[1575] := 25, Buffer[1577] := 25, Buffer[1581] := 25, Buffer[1586] := 15, Buffer[1587] := -125, Buffer[1588] := -20, Buffer[1589] := -95, Buffer[1590] := 50,
        Buffer[1591] := 54, Buffer[1592] := 48, Buffer[1593] := 51, Buffer[1594] := 48, Buffer[1595] := 52, Buffer[1596] := 48, Buffer[1597] := 51, Buffer[1598] := 51, Buffer[1613] := 93, Buffer[1615] := -115, Buffer[1616] := 2, Buffer[1617] := 89, Buffer[1618] := 19, Buffer[1619] := -119, Buffer[1622] := 29, Buffer[1623] := -75, Buffer[1626] := 29, Buffer[1627] := -15, Buffer[1628] := 7, Buffer[1629] := -41, Buffer[1631] := 60, Buffer[1632] := 107, Buffer[1633] := 99, Buffer[1634] := 111, Buffer[1641] := 3, Buffer[1643] := 25, Buffer[1645] := 25, Buffer[1649] := 25, Buffer[1654] := 15, Buffer[1655] := -125, Buffer[1656] := -20, Buffer[1657] := -95, Buffer[1658] := 50, Buffer[1659] := 54, Buffer[1660] := 48, Buffer[1661] := 51, Buffer[1662] := 48, Buffer[1663] := 52, Buffer[1664] := 48, Buffer[1665] := 51, Buffer[1666] := 51, Buffer[1681] := 93, Buffer[1683] := -115, Buffer[1684] := 2, Buffer[1685] := 89, Buffer[1686] := 19, Buffer[1687] := -119, Buffer[1690] := 29, Buffer[1691] := -75, Buffer[1694] := 29, Buffer[1695] := -15, Buffer[1696] := 7, Buffer[1697] := -41, Buffer[1699] := 60, Buffer[1700] := 107, Buffer[1701] := 99, Buffer[1702] := 111, Buffer[1709] := 3, Buffer[1711] := 25, Buffer[1713] := 39,
        Buffer[1717] := 39, Buffer[1722] := 15, Buffer[1723] := -125, Buffer[1724] := -20, Buffer[1725] := -104, Buffer[1726] := 50, Buffer[1727] := 54, Buffer[1728] := 48, Buffer[1729] := 51, Buffer[1730] := 48, Buffer[1731] := 52, Buffer[1732] := 48, Buffer[1733] := 50, Buffer[1734] := 52, Buffer[1749] := 94, Buffer[1751] := -115, Buffer[1752] := 2, Buffer[1753] := 88, Buffer[1754] := 20, Buffer[1755] := 80, Buffer[1758] := 36, Buffer[1759] := 37, Buffer[1762] := 36, Buffer[1763] := 97, Buffer[1764] := 7, Buffer[1765] := -43, Buffer[1767] := 60, Buffer[1768] := 107, Buffer[1769] := 99, Buffer[1770] := 111, Buffer[1777] := 2, Buffer[1779] := 42, Buffer[1781] := 39, Buffer[1785] := 39, Buffer[1790] := 15, Buffer[1791] := -125, Buffer[1792] := -20, Buffer[1793] := -104, Buffer[1794] := 50, Buffer[1795] := 54, Buffer[1796] := 48, Buffer[1797] := 51, Buffer[1798] := 48, Buffer[1799] := 52, Buffer[1800] := 48, Buffer[1801] := 50, Buffer[1802] := 52, Buffer[1817] := 94, Buffer[1819] := -115, Buffer[1820] := 2, Buffer[1821] := 88, Buffer[1822] := 20, Buffer[1823] := 80, Buffer[1826] := 36, Buffer[1827] := 37, Buffer[1830] := 36, Buffer[1831] := 97, Buffer[1832] := 7, Buffer[1833] := -43, Buffer[1835] := 60,
        Buffer[1836] := 107, Buffer[1837] := 99, Buffer[1838] := 111, Buffer[1845] := 2, Buffer[1847] := 43, Buffer[1849] := 40, Buffer[1853] := 40, Buffer[1858] := 15, Buffer[1859] := -125, Buffer[1860] := -20, Buffer[1861] := -104, Buffer[1862] := 50, Buffer[1863] := 54, Buffer[1864] := 48, Buffer[1865] := 51, Buffer[1866] := 48, Buffer[1867] := 52, Buffer[1868] := 48, Buffer[1869] := 50, Buffer[1870] := 52, Buffer[1885] := -115, Buffer[1887] := 55, Buffer[1888] := 20, Buffer[1889] := 80, Buffer[1890] := 1, Buffer[1891] := -112, Buffer[1894] := 26, Buffer[1895] := 122, Buffer[1898] := 26, Buffer[1899] := -74, Buffer[1900] := 7, Buffer[1901] := -42, Buffer[1903] := 60, Buffer[1904] := 107, Buffer[1905] := 99, Buffer[1906] := 111, Buffer[1913] := 2, Buffer[1915] := 56, Buffer[1917] := 40, Buffer[1921] := 40, Buffer[1926] := 15, Buffer[1927] := -125, Buffer[1928] := -20, Buffer[1929] := -114, Buffer[1930] := 50, Buffer[1931] := 54, Buffer[1932] := 48, Buffer[1933] := 51, Buffer[1934] := 48, Buffer[1935] := 52, Buffer[1936] := 48, Buffer[1937] := 49, Buffer[1938] := 52, Buffer[1953] := 53, Buffer[1955] := 95, Buffer[1956] := 1, Buffer[1957] := -112, Buffer[1958] := 2, Buffer[1959] := 89, Buffer[1962] := 19,
        Buffer[1963] := -5, Buffer[1966] := 20, Buffer[1967] := 55, Buffer[1968] := 7, Buffer[1969] := -41, Buffer[1971] := 60, Buffer[1972] := 107, Buffer[1973] := 99, Buffer[1974] := 111, Buffer[1981] := 2, Buffer[1983] := 93, Buffer[1985] := 32, Buffer[1989] := 32, Buffer[1994] := 15, Buffer[1995] := -125, Buffer[1996] := -24, Buffer[1997] := -64, Buffer[1998] := 50, Buffer[1999] := 54, Buffer[2000] := 48, Buffer[2001] := 51, Buffer[2002] := 48, Buffer[2003] := 51, Buffer[2004] := 48, Buffer[2005] := 52, Buffer[2006] := 48, Buffer[2021] := 81, Buffer[2023] := 93, Buffer[2024] := 1, Buffer[2025] := 44, Buffer[2026] := 2, Buffer[2027] := 88, Buffer[2030] := 13, Buffer[2031] := 70, Buffer[2034] := 13, Buffer[2035] := -126, Buffer[2036] := 7, Buffer[2037] := -44, Buffer[2039] := 60, Buffer[2040] := 107, Buffer[2041] := 99, Buffer[2042] := 111, Buffer[2049] := 2, Buffer[2051] := 93, Buffer[2053] := 32, Buffer[2057] := 32, Buffer[2062] := 15, Buffer[2063] := -125, Buffer[2064] := -24, Buffer[2065] := -64, Buffer[2066] := 50, Buffer[2067] := 54, Buffer[2068] := 48, Buffer[2069] := 51, Buffer[2070] := 48, Buffer[2071] := 51, Buffer[2072] := 48, Buffer[2073] := 52, Buffer[2074] := 48, Buffer[2089] := 81,
        Buffer[2091] := 93, Buffer[2092] := 1, Buffer[2093] := 44, Buffer[2094] := 2, Buffer[2095] := 88, Buffer[2098] := 13, Buffer[2099] := 70, Buffer[2102] := 13, Buffer[2103] := -126, Buffer[2104] := 7, Buffer[2105] := -44, Buffer[2107] := 60, Buffer[2108] := 107, Buffer[2109] := 99, Buffer[2110] := 111, Buffer[2117] := 2, Buffer[2119] := 93, Buffer[2121] := 32, Buffer[2125] := 32, Buffer[2130] := 15, Buffer[2131] := -125, Buffer[2132] := -24, Buffer[2133] := -64, Buffer[2134] := 50, Buffer[2135] := 54, Buffer[2136] := 48, Buffer[2137] := 51, Buffer[2138] := 48, Buffer[2139] := 51, Buffer[2140] := 48, Buffer[2141] := 52, Buffer[2142] := 48, Buffer[2157] := 81, Buffer[2159] := 93, Buffer[2160] := 1, Buffer[2161] := 44, Buffer[2162] := 2, Buffer[2163] := 88, Buffer[2166] := 13, Buffer[2167] := 70, Buffer[2170] := 13, Buffer[2171] := -126, Buffer[2172] := 7, Buffer[2173] := -44, Buffer[2175] := 60, Buffer[2178] := 13, Buffer[2179] := 70, Buffer[2182] := 13, Buffer[2183] := -126, Buffer[2184] := 7, Buffer[2185] := -44, Buffer[2187] := 60, Buffer[2189] := 55, Buffer[2193] := 55, Buffer[2198] := 15, Buffer[2199] := -125, Buffer[2200] := -20, Buffer[2201] := -119, Buffer[2202] := 50, Buffer[2203] := 54,
        Buffer[2204] := 48, Buffer[2205] := 51, Buffer[2206] := 48, Buffer[2207] := 52, Buffer[2208] := 48, Buffer[2209] := 48, Buffer[2210] := 57, Buffer[2225] := 55, Buffer[2227] := 94, Buffer[2228] := 1, Buffer[2229] := -112, Buffer[2230] := 2, Buffer[2231] := 88, Buffer[2234] := 24, Buffer[2235] := -92, Buffer[2238] := 24, Buffer[2239] := -32, Buffer[2240] := 7, Buffer[2241] := -45, Buffer[2243] := 60, Buffer[2244] := 107, Buffer[2245] := 99, Buffer[2246] := 111, Buffer[2253] := 2, Buffer[2255] := 97, Buffer[2257] := 55, Buffer[2261] := 55, Buffer[2266] := 15, Buffer[2267] := -125, Buffer[2268] := -20, Buffer[2269] := -119, Buffer[2270] := 50, Buffer[2271] := 54, Buffer[2272] := 48, Buffer[2273] := 51, Buffer[2274] := 48, Buffer[2275] := 52, Buffer[2276] := 48, Buffer[2277] := 48, Buffer[2278] := 57, Buffer[2293] := 55, Buffer[2295] := 94, Buffer[2296] := 1, Buffer[2297] := -112, Buffer[2298] := 2, Buffer[2299] := 88, Buffer[2302] := 24, Buffer[2303] := -92, Buffer[2306] := 24, Buffer[2307] := -32, Buffer[2308] := 7, Buffer[2309] := -45, Buffer[2311] := 60, Buffer[2312] := 107, Buffer[2313] := 99, Buffer[2314] := 111, Buffer[2321] := 2, Buffer[2323] := 97, Buffer[2325] := 55, Buffer[2329] := 55,
        Buffer[2334] := 15, Buffer[2335] := -125, Buffer[2336] := -20, Buffer[2337] := -119, Buffer[2338] := 50, Buffer[2339] := 54, Buffer[2340] := 48, Buffer[2341] := 51, Buffer[2342] := 48, Buffer[2343] := 52, Buffer[2344] := 48, Buffer[2345] := 48, Buffer[2346] := 57, Buffer[2361] := 55, Buffer[2363] := 94, Buffer[2364] := 1, Buffer[2365] := -112, Buffer[2366] := 2, Buffer[2367] := 88, Buffer[2370] := 24, Buffer[2371] := -92, Buffer[2374] := 24, Buffer[2375] := -32, Buffer[2376] := 7, Buffer[2377] := -45, Buffer[2379] := 60, Buffer[2380] := 107, Buffer[2381] := 99, Buffer[2382] := 111, Buffer[2389] := 2, Buffer[2391] := 97, Buffer[2393] := 55, Buffer[2397] := 55, Buffer[2402] := 15, Buffer[2403] := -125, Buffer[2404] := -20, Buffer[2405] := -119, Buffer[2406] := 50, Buffer[2407] := 54, Buffer[2408] := 48, Buffer[2409] := 51, Buffer[2410] := 48, Buffer[2411] := 52, Buffer[2412] := 48, Buffer[2413] := 48, Buffer[2414] := 57, Buffer[2429] := 55, Buffer[2431] := 94, Buffer[2432] := 1, Buffer[2433] := -112, Buffer[2434] := 2, Buffer[2435] := 88, Buffer[2438] := 24, Buffer[2439] := -92, Buffer[2442] := 24, Buffer[2443] := -32, Buffer[2444] := 7, Buffer[2445] := -45, Buffer[2447] := 60, Buffer[2448] := 107,
        Buffer[2449] := 99, Buffer[2450] := 111, Buffer[2457] := 2, Buffer[2459] := 63, Buffer[2461] := 42, Buffer[2465] := 42, Buffer[2470] := 15, Buffer[2471] := -126, Buffer[2472] := -72, Buffer[2473] := 15, Buffer[2474] := 50, Buffer[2475] := 54, Buffer[2476] := 48, Buffer[2477] := 50, Buffer[2478] := 50, Buffer[2479] := 53, Buffer[2480] := 48, Buffer[2481] := 51, Buffer[2482] := 57, Buffer[2497] := -115, Buffer[2499] := 55, Buffer[2500] := 19, Buffer[2501] := -20, Buffer[2502] := 1, Buffer[2503] := -112, Buffer[2506] := 42, Buffer[2507] := 71, Buffer[2510] := 42, Buffer[2511] := -125, Buffer[2512] := 7, Buffer[2513] := -45, Buffer[2515] := 60, Buffer[2516] := 107, Buffer[2517] := 99, Buffer[2518] := 111, Buffer[2525] := 2, Buffer[2527] := 63, Buffer[2529] := 42, Buffer[2533] := 42, Buffer[2538] := 15, Buffer[2539] := -126, Buffer[2540] := -72, Buffer[2541] := 15, Buffer[2542] := 50, Buffer[2543] := 54, Buffer[2544] := 48, Buffer[2545] := 50, Buffer[2546] := 50, Buffer[2547] := 53, Buffer[2548] := 48, Buffer[2549] := 51, Buffer[2550] := 57, Buffer[2565] := -115, Buffer[2567] := 55, Buffer[2568] := 19, Buffer[2569] := -20, Buffer[2570] := 1, Buffer[2571] := -112, Buffer[2574] := 42, Buffer[2575] := 71,
        Buffer[2578] := 42, Buffer[2579] := -125, Buffer[2580] := 7, Buffer[2581] := -45, Buffer[2583] := 60, Buffer[2584] := 107, Buffer[2585] := 99, Buffer[2586] := 111, Buffer[2593] := 2, Buffer[2595] := 63, Buffer[2597] := 42, Buffer[2601] := 42, Buffer[2606] := 15, Buffer[2607] := -126, Buffer[2608] := -72, Buffer[2609] := 15, Buffer[2610] := 50, Buffer[2611] := 54, Buffer[2612] := 48, Buffer[2613] := 50, Buffer[2614] := 50, Buffer[2615] := 53, Buffer[2616] := 48, Buffer[2617] := 51, Buffer[2618] := 57, Buffer[2633] := -115, Buffer[2635] := 55, Buffer[2636] := 19, Buffer[2637] := -20, Buffer[2638] := 1, Buffer[2639] := -112, Buffer[2642] := 42, Buffer[2643] := 71, Buffer[2646] := 42, Buffer[2647] := -125, Buffer[2648] := 7, Buffer[2649] := -45, Buffer[2651] := 60, Buffer[2652] := 107, Buffer[2653] := 99, Buffer[2654] := 111, Buffer[2661] := 2, Buffer[2663] := 63, Buffer[2665] := 42, Buffer[2669] := 42, Buffer[2674] := 15, Buffer[2675] := -126, Buffer[2676] := -72, Buffer[2677] := 15, Buffer[2678] := 50, Buffer[2679] := 54, Buffer[2680] := 48, Buffer[2681] := 50, Buffer[2682] := 50, Buffer[2683] := 53, Buffer[2684] := 48, Buffer[2685] := 51, Buffer[2686] := 57, Buffer[2701] := -115, Buffer[2703] := 55,
        Buffer[2704] := 19, Buffer[2705] := -20, Buffer[2706] := 1, Buffer[2707] := -112, Buffer[2710] := 42, Buffer[2711] := 71, Buffer[2714] := 42, Buffer[2715] := -125, Buffer[2716] := 7, Buffer[2717] := -45, Buffer[2719] := 60, Buffer[2720] := 107, Buffer[2721] := 99, Buffer[2722] := 111, Buffer[2729] := 2, Buffer[2731] := 63, Buffer[2733] := 42, Buffer[2737] := 42, Buffer[2742] := 15, Buffer[2743] := -126, Buffer[2744] := -72, Buffer[2745] := 15, Buffer[2746] := 50, Buffer[2747] := 54, Buffer[2748] := 48, Buffer[2749] := 50, Buffer[2750] := 50, Buffer[2751] := 53, Buffer[2752] := 48, Buffer[2753] := 51, Buffer[2754] := 57, Buffer[2769] := -115, Buffer[2771] := 55, Buffer[2772] := 19, Buffer[2773] := -20, Buffer[2774] := 1, Buffer[2775] := -112, Buffer[2778] := 42, Buffer[2779] := 71, Buffer[2782] := 42, Buffer[2783] := -125, Buffer[2784] := 7, Buffer[2785] := -45, Buffer[2787] := 60, Buffer[2788] := 107, Buffer[2789] := 99, Buffer[2790] := 111, Buffer[2797] := 2, Buffer[2799] := 68, Buffer[2801] := 65, Buffer[2805] := 65, Buffer[2810] := 15, Buffer[2811] := -126, Buffer[2812] := -76, Buffer[2813] := 46, Buffer[2814] := 50, Buffer[2815] := 54, Buffer[2816] := 48, Buffer[2817] := 50, Buffer[2818] := 50,
        Buffer[2819] := 52, Buffer[2820] := 48, Buffer[2821] := 52, Buffer[2822] := 54, Buffer[2837] := 66, Buffer[2839] := 95, Buffer[2840] := 1, Buffer[2841] := -12, Buffer[2842] := 2, Buffer[2843] := 88, Buffer[2846] := 35, Buffer[2847] := -100, Buffer[2850] := 35, Buffer[2851] := -40, Buffer[2852] := 7, Buffer[2853] := -42, Buffer[2855] := 60, Buffer[2856] := 107, Buffer[2857] := 99, Buffer[2858] := 111, Buffer[2865] := 2, Buffer[2867] := 68, Buffer[2869] := 65, Buffer[2873] := 65, Buffer[2878] := 15, Buffer[2879] := -126, Buffer[2880] := -76, Buffer[2881] := 46, Buffer[2882] := 50, Buffer[2883] := 54, Buffer[2884] := 48, Buffer[2885] := 50, Buffer[2886] := 50, Buffer[2887] := 52, Buffer[2888] := 48, Buffer[2889] := 52, Buffer[2890] := 54, Buffer[2905] := 66, Buffer[2907] := 95, Buffer[2908] := 1, Buffer[2909] := -12, Buffer[2910] := 2, Buffer[2911] := 88, Buffer[2914] := 35, Buffer[2915] := -100, Buffer[2918] := 35, Buffer[2919] := -40, Buffer[2920] := 7, Buffer[2921] := -42, Buffer[2923] := 60, Buffer[2924] := 107, Buffer[2925] := 99, Buffer[2926] := 111, Buffer[2933] := 2, Buffer[2935] := 102, Buffer[2937] := 92, Buffer[2941] := 92, Buffer[2946] := 15, Buffer[2947] := -126, Buffer[2948] := 121,
        Buffer[2949] := -124, Buffer[2950] := 50, Buffer[2951] := 54, Buffer[2952] := 48, Buffer[2953] := 50, Buffer[2954] := 48, Buffer[2955] := 57, Buffer[2956] := 48, Buffer[2957] := 50, Buffer[2958] := 56, Buffer[2973] := 94, Buffer[2975] := -115, Buffer[2976] := 2, Buffer[2977] := 89, Buffer[2978] := 19, Buffer[2979] := -119, Buffer[2982] := 49, Buffer[2983] := -126, Buffer[2986] := 49, Buffer[2987] := -66, Buffer[2988] := 7, Buffer[2989] := -39, Buffer[2991] := 60, Buffer[2992] := 107, Buffer[2993] := 99, Buffer[2994] := 111, Buffer[3001] := 2, Buffer[3003] := -128, Buffer[3005] := 79, Buffer[3009] := 79, Buffer[3014] := 15, Buffer[3015] := -127, Buffer[3016] := 25, Buffer[3017] := -29, Buffer[3018] := 50, Buffer[3019] := 54, Buffer[3020] := 48, Buffer[3021] := 49, Buffer[3022] := 49, Buffer[3023] := 57, Buffer[3024] := 48, Buffer[3025] := 49, Buffer[3026] := 49, Buffer[3041] := 55, Buffer[3043] := 91, Buffer[3044] := 1, Buffer[3045] := -112, Buffer[3046] := 2, Buffer[3047] := 88, Buffer[3050] := 36, Buffer[3051] := -9, Buffer[3054] := 37, Buffer[3055] := 51, Buffer[3056] := 7, Buffer[3057] := -44, Buffer[3059] := 60, Buffer[3060] := 48, Buffer[3061] := 52, Buffer[3062] := 52, Buffer[3077] := 57,
        Buffer[3079] := 95, Buffer[3080] := 1, Buffer[3081] := -112, Buffer[3082] := 2, Buffer[3083] := 88, Buffer[3086] := 21, Buffer[3087] := -105, Buffer[3090] := 21, Buffer[3091] := -45, Buffer[3092] := 7, Buffer[3093] := -43, Buffer[3095] := 60, Buffer[3096] := 107, Buffer[3097] := 99, Buffer[3098] := 111, Buffer[3105] := 2, Buffer[3107] := 26, Buffer[3109] := 20, Buffer[3113] := 20, Buffer[3118] := 15, Buffer[3119] := -127, Buffer[3120] := 6, Buffer[3121] := 126, Buffer[3122] := 50, Buffer[3123] := 54, Buffer[3124] := 48, Buffer[3125] := 49, Buffer[3126] := 49, Buffer[3127] := 52, Buffer[3128] := 48, Buffer[3129] := 52, Buffer[3130] := 54, Buffer[3145] := 58, Buffer[3147] := 65, Buffer[3148] := 1, Buffer[3149] := -112, Buffer[3150] := 1, Buffer[3151] := -12, Buffer[3154] := 22, Buffer[3155] := 73, Buffer[3158] := 22, Buffer[3159] := -123, Buffer[3160] := 7, Buffer[3161] := -43, Buffer[3163] := 60, Buffer[3164] := 107, Buffer[3165] := 99, Buffer[3166] := 111, Buffer[3173] := 2, Buffer[3175] := 26, Buffer[3177] := 21, Buffer[3181] := 21, Buffer[3186] := 15, Buffer[3187] := -127, Buffer[3188] := 6, Buffer[3189] := 124, Buffer[3190] := 50, Buffer[3191] := 54, Buffer[3192] := 48, Buffer[3193] := 49,
        Buffer[3194] := 49, Buffer[3195] := 52, Buffer[3196] := 48, Buffer[3197] := 52, Buffer[3198] := 52, Buffer[3213] := 95, Buffer[3215] := -115, Buffer[3216] := 2, Buffer[3217] := 88, Buffer[3218] := 20, Buffer[3219] := 80, Buffer[3222] := 28, Buffer[3223] := -37, Buffer[3226] := 29, Buffer[3227] := 23, Buffer[3228] := 7, Buffer[3229] := -42, Buffer[3231] := 60, Buffer[3232] := 107, Buffer[3233] := 99, Buffer[3234] := 111, Buffer[3241] := 2, Buffer[3243] := 26, Buffer[3245] := 22, Buffer[3249] := 22, Buffer[3254] := 15, Buffer[3255] := -127, Buffer[3256] := 6, Buffer[3257] := 124, Buffer[3258] := 50, Buffer[3259] := 54, Buffer[3260] := 48, Buffer[3261] := 49, Buffer[3262] := 49, Buffer[3263] := 52, Buffer[3264] := 48, Buffer[3265] := 52, Buffer[3266] := 52, Buffer[3281] := -115, Buffer[3283] := 63, Buffer[3284] := 20, Buffer[3285] := 80, Buffer[3286] := 1, Buffer[3287] := -12, Buffer[3290] := 29, Buffer[3291] := 33, Buffer[3294] := 29, Buffer[3295] := 93, Buffer[3296] := 7, Buffer[3297] := -41, Buffer[3299] := 60, Buffer[3300] := 107, Buffer[3301] := 99, Buffer[3302] := 111, Buffer[3309] := 2, Buffer[3311] := 26, Buffer[3313] := 23, Buffer[3317] := 23, Buffer[3322] := 15, Buffer[3323] := -127,
        Buffer[3324] := 6, Buffer[3325] := 126, Buffer[3326] := 50, Buffer[3327] := 54, Buffer[3328] := 48, Buffer[3329] := 49, Buffer[3330] := 49, Buffer[3331] := 52, Buffer[3332] := 48, Buffer[3333] := 52, Buffer[3334] := 54, Buffer[3349] := 65, Buffer[3351] := 94, Buffer[3352] := 1, Buffer[3353] := -12, Buffer[3354] := 2, Buffer[3355] := 88, Buffer[3358] := 32, Buffer[3359] := 105, Buffer[3362] := 32, Buffer[3363] := -91, Buffer[3364] := 7, Buffer[3365] := -42, Buffer[3367] := 60, Buffer[3368] := 107, Buffer[3369] := 99, Buffer[3370] := 111, Buffer[3377] := 2, Buffer[3379] := 26, Buffer[3381] := 24, Buffer[3385] := 24, Buffer[3390] := 15, Buffer[3391] := -127, Buffer[3392] := 6, Buffer[3393] := 124, Buffer[3394] := 50, Buffer[3395] := 54, Buffer[3396] := 48, Buffer[3397] := 49, Buffer[3398] := 49, Buffer[3399] := 52, Buffer[3400] := 48, Buffer[3401] := 52, Buffer[3402] := 52, Buffer[3417] := 63, Buffer[3419] := 95, Buffer[3420] := 1, Buffer[3421] := -12, Buffer[3422] := 2, Buffer[3423] := 89, Buffer[3426] := 37, Buffer[3427] := 37, Buffer[3430] := 37, Buffer[3431] := 97, Buffer[3432] := 7, Buffer[3433] := -40, Buffer[3435] := 60, Buffer[3436] := 107, Buffer[3437] := 99, Buffer[3438] := 111,
        Buffer[3445] := 2, Buffer[3447] := 26, Buffer[3449] := 25, Buffer[3453] := 25, Buffer[3458] := 15, Buffer[3459] := -127, Buffer[3460] := 6, Buffer[3461] := 126, Buffer[3462] := 50, Buffer[3463] := 54, Buffer[3464] := 48, Buffer[3465] := 49, Buffer[3466] := 49, Buffer[3467] := 52, Buffer[3468] := 48, Buffer[3469] := 52, Buffer[3470] := 54, Buffer[3485] := 94, Buffer[3487] := -115, Buffer[3488] := 2, Buffer[3489] := 88, Buffer[3490] := 19, Buffer[3491] := -119, Buffer[3494] := 39, Buffer[3495] := -83, Buffer[3498] := 39, Buffer[3499] := -23, Buffer[3500] := 7, Buffer[3501] := -41, Buffer[3503] := 60, Buffer[3504] := 107, Buffer[3505] := 99, Buffer[3506] := 111, Buffer[3513] := 2, Buffer[3515] := 26, Buffer[3517] := 26, Buffer[3521] := 26, Buffer[3526] := 15, Buffer[3527] := -127, Buffer[3528] := 6, Buffer[3529] := 124, Buffer[3530] := 50, Buffer[3531] := 54, Buffer[3532] := 48, Buffer[3533] := 49, Buffer[3534] := 49, Buffer[3535] := 52, Buffer[3536] := 48, Buffer[3537] := 52, Buffer[3538] := 52, Buffer[3553] := 95, Buffer[3555] := -115, Buffer[3556] := 2, Buffer[3557] := 89, Buffer[3558] := 19, Buffer[3559] := -119, Buffer[3562] := 44, Buffer[3563] := 105, Buffer[3566] := 44, Buffer[3567] := -91,
        Buffer[3568] := 7, Buffer[3569] := -39, Buffer[3571] := 60, Buffer[3572] := 107, Buffer[3573] := 99, Buffer[3574] := 111, Buffer[3581] := 3, Buffer[3583] := 26, Buffer[3597] := 55, Buffer[3599] := 91, Buffer[3600] := 1, Buffer[3601] := -112, Buffer[3602] := 2, Buffer[3603] := 89, Buffer[3606] := 34, Buffer[3607] := 30, Buffer[3610] := 34, Buffer[3611] := 90, Buffer[3612] := 7, Buffer[3613] := -41, Buffer[3615] := 60, Buffer[3616] := 107, Buffer[3617] := 99, Buffer[3618] := 111, Buffer[3625] := 2, Buffer[3627] := 84, Buffer[3629] := 54, Buffer[3633] := 54, Buffer[3638] := 15, Buffer[3639] := -127, Buffer[3640] := 6, Buffer[3641] := 108, Buffer[3642] := 50, Buffer[3643] := 54, Buffer[3644] := 48, Buffer[3645] := 49, Buffer[3646] := 49, Buffer[3647] := 52, Buffer[3648] := 48, Buffer[3649] := 50, Buffer[3650] := 56, Buffer[3665] := 91, Buffer[3667] := -115, Buffer[3668] := 2, Buffer[3669] := 89, Buffer[3670] := 19, Buffer[3671] := -119, Buffer[3674] := 34, Buffer[3675] := 90, Buffer[3678] := 34, Buffer[3679] := -106, Buffer[3680] := 7, Buffer[3681] := -40, Buffer[3683] := 60, Buffer[3684] := 107, Buffer[3685] := 99, Buffer[3686] := 111, Buffer[3693] := 2, Buffer[3695] := 84, Buffer[3697] := 55,
        Buffer[3701] := 55, Buffer[3706] := 15, Buffer[3707] := -127, Buffer[3708] := 6, Buffer[3709] := 103, Buffer[3710] := 50, Buffer[3711] := 54, Buffer[3712] := 48, Buffer[3713] := 49, Buffer[3714] := 49, Buffer[3715] := 52, Buffer[3716] := 48, Buffer[3717] := 50, Buffer[3718] := 51, Buffer[3733] := 95, Buffer[3735] := -115, Buffer[3736] := 2, Buffer[3737] := 88, Buffer[3738] := 19, Buffer[3739] := -119, Buffer[3742] := 35, Buffer[3743] := 23, Buffer[3746] := 35, Buffer[3747] := 83, Buffer[3748] := 7, Buffer[3749] := -43, Buffer[3751] := 60, Buffer[3752] := 107, Buffer[3753] := 99, Buffer[3754] := 111, Buffer[3761] := 2, Buffer[3763] := 84, Buffer[3765] := 56, Buffer[3769] := 56, Buffer[3774] := 15, Buffer[3775] := -127, Buffer[3776] := 6, Buffer[3777] := 115, Buffer[3778] := 50, Buffer[3779] := 54, Buffer[3780] := 48, Buffer[3781] := 49, Buffer[3782] := 49, Buffer[3783] := 52, Buffer[3784] := 48, Buffer[3785] := 51, Buffer[3786] := 53, Buffer[3801] := 26, Buffer[3803] := -115, Buffer[3805] := -6, Buffer[3806] := 19, Buffer[3807] := -20, Buffer[3810] := 36, Buffer[3811] := 20, Buffer[3814] := 36, Buffer[3815] := 80, Buffer[3816] := 7, Buffer[3817] := -46, Buffer[3819] := 60, Buffer[3820] := 107,
        Buffer[3821] := 99, Buffer[3822] := 111, Buffer[3829] := 2, Buffer[3831] := 84, Buffer[3833] := 57, Buffer[3837] := 57, Buffer[3842] := 15, Buffer[3843] := -127, Buffer[3844] := 6, Buffer[3845] := 115, Buffer[3846] := 50, Buffer[3847] := 54, Buffer[3848] := 48, Buffer[3849] := 49, Buffer[3850] := 49, Buffer[3851] := 52, Buffer[3852] := 48, Buffer[3853] := 51, Buffer[3854] := 53, Buffer[3869] := -115, Buffer[3871] := 56, Buffer[3872] := 19, Buffer[3873] := -20, Buffer[3874] := 1, Buffer[3875] := -112, Buffer[3878] := 36, Buffer[3879] := 90, Buffer[3882] := 36, Buffer[3883] := -106, Buffer[3884] := 7, Buffer[3885] := -45, Buffer[3887] := 60, Buffer[3888] := 107, Buffer[3889] := 99, Buffer[3890] := 111, Buffer[3897] := 2, Buffer[3899] := 84);   // Data Bloc Receive from OPTP
   Read_Request : BOOL;
   Swapp_buf : BOOL;
   trigger_Co : BOOL := 1;
   trigger_Del : BOOL;
   Write_Request : BOOL;
END_VAR

ROUTINE _01_00_Connection_Management   (* ladder *)
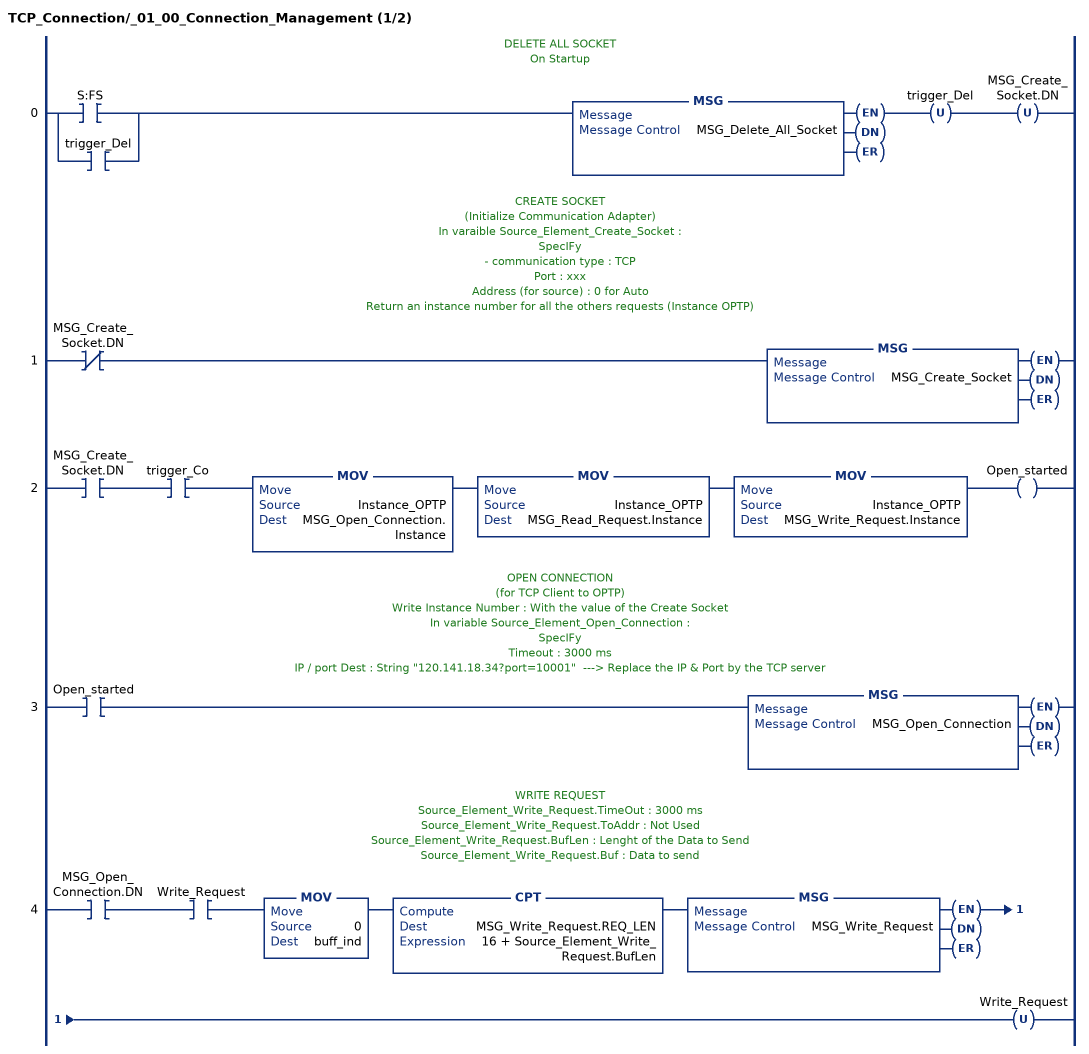
   // DELETE ALL SOCKET
   // On Startup
   0: [XIC(S:FS) ,XIC(trigger_Del) ]MSG(MSG_Delete_All_Socket)OTU(trigger_Del)OTU(MSG_Create_Socket.DN);
   // CREATE SOCKET
   // (Initialize Communication Adapter)
   // In varaible Source_Element_Create_Socket :
   // SpecIFy
   // - communication type : TCP
   // Port : xxx
   // Address (for source) : 0 for Auto
   // Return an instance number for all the others requests (Instance OPTP)
   1: XIO(MSG_Create_Socket.DN)MSG(MSG_Create_Socket);
   2: XIC(MSG_Create_Socket.DN)XIC(trigger_Co)MOV(Instance_OPTP,MSG_Open_Connection.Instance)MOV(Instance_OPTP,MSG_Read_Request.Instance)MOV(Instance_OPTP,MSG_Write_Request.Instance)OTE(Open_started);
   // OPEN CONNECTION
   // (for TCP Client to OPTP)
   // Write Instance Number : With the value of the Create Socket
   // In variable Source_Element_Open_Connection :
   // SpecIFy
   // Timeout : 3000 ms
   // IP / port Dest : String "120.141.18.34?port=10001"  ---> Replace the IP & Port by the TCP server
   3: XIC(Open_started)MSG(MSG_Open_Connection);
   // WRITE REQUEST
   //  Source_Element_Write_Request.TimeOut : 3000 ms
   // Source_Element_Write_Request.ToAddr : Not Used
   // Source_Element_Write_Request.BufLen : Lenght of the Data to Send
   // Source_Element_Write_Request.Buf : Data to send
   4: XIC(MSG_Open_Connection.DN)XIC(Write_Request)MOV(0,buff_ind)CPT(MSG_Write_Request.REQ_LEN,16 + Source_Element_Write_Request.BufLen)MSG(MSG_Write_Request)OTU(Write_Request);
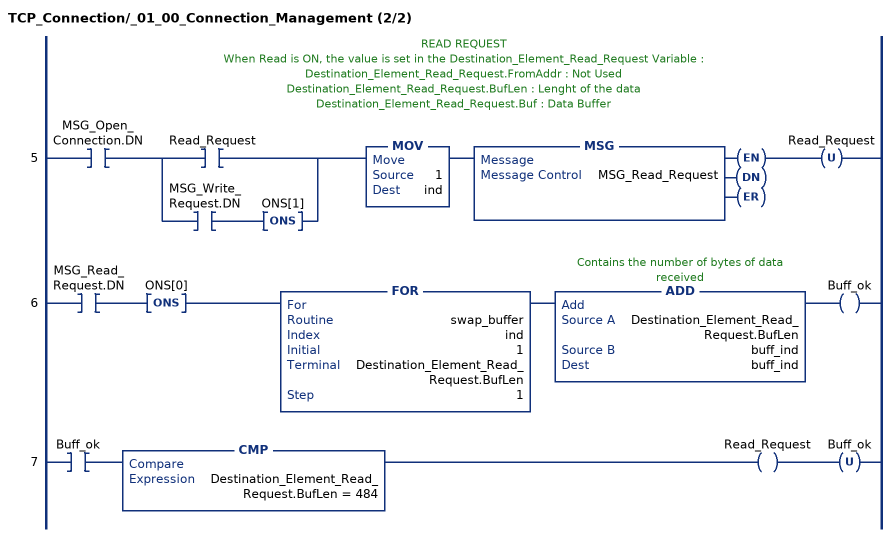
   // READ REQUEST
   //  When Read is ON, the value is set in the Destination_Element_Read_Request Variable :
   // Destination_Element_Read_Request.FromAddr : Not Used
   // Destination_Element_Read_Request.BufLen : Lenght of the data
   // Destination_Element_Read_Request.Buf : Data Buffer
   5: XIC(MSG_Open_Connection.DN)[XIC(Read_Request) ,XIC(MSG_Write_Request.DN) ONS(ONS[1]) ]MOV(1,ind)MSG(MSG_Read_Request)OTU(Read_Request);
   6: XIC(MSG_Read_Request.DN)ONS(ONS[0])FOR(swap_buffer,ind,1,Destination_Element_Read_Request.BufLen,1)ADD(Destination_Element_Read_Request.BufLen,buff_ind,buff_ind)OTE(Buff_ok);
   7: XIC(Buff_ok)CMP(Destination_Element_Read_Request.BufLen = 484)OTE(Read_Request)OTU(Buff_ok);
END_ROUTINE

ROUTINE Main   (* ladder *)
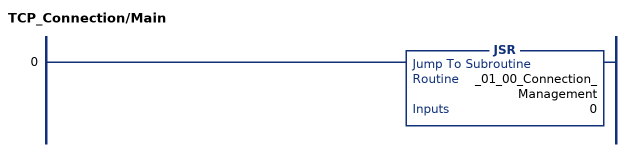
   0: JSR(_01_00_Connection_Management,0);
END_ROUTINE

ROUTINE swap_buffer   (* ladder *)
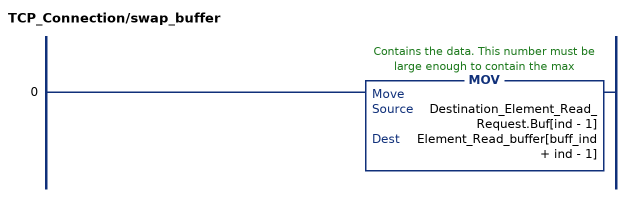
   0: MOV(Destination_Element_Read_Request.Buf[ind - 1],Element_Read_buffer[buff_ind + ind - 1]);
END_ROUTINE
END_PROGRAM
